// TIA Portal V21 export
FUNCTION_BLOCK "FB307"   // FB307, LAD
TITLE = FB307
{ S7_Optimized_Access := 'FALSE' }
AUTHOR : PRECISE
FAMILY : PRECISE
// RAW MATERIAL ADDITION MANUAL
// stored: AutoNumber false, SetENOAutomatically false
   VAR_INPUT
      Enable : Bool;
      Disable : Bool;
      Fault : Bool;
      SecPulse : Bool;
      AlwaysTrue : Bool;
      StartConfirmationPopupSel : Bool;   // StartConfirmationPopupSel: 0-NO/1-YES
      EndConfirmationPopupSel : Bool;   // EndConfirmationPopupSel: 0-NO/1-YES
      MixingTimerDone : Bool;
      SetRMNo : Int := 1;   // Max-10
      VesselSafetyPressure : Real;
      VesselActPressure : Real;
   END_VAR
   VAR_OUTPUT
      StartConfirmationPopup : Bool;   // For Start Confirmation Popup Selection: Yes
      EndConfirmationPopup : Bool;   // For End Confirmation Popup Selection: Yes
      RMAddPopup : Bool;
      VisibleRM1 : Bool;
      VisibleRM2 : Bool;
      VisibleRM3 : Bool;
      VisibleRM4 : Bool;
      VisibleRM5 : Bool;
      VisibleRM6 : Bool;
      VisibleRM7 : Bool;
      VisibleRM8 : Bool;
      VisibleRM9 : Bool;
      VisibleRM10 : Bool;
      PrintTrigger : Bool;
      MixerCmd : Bool;
      PrintWord : Int;
      PrintStatus : String[50];
      VesselUnderPressure : Bool;
   END_VAR
   VAR_IN_OUT
      Start : Bool;
      Stop : Bool;
      Reset : Bool;
      StartConfirmationAck : Bool;   // For Start Confirmation Popup Selection: Yes
      EndConfirmationAck : Bool;   // For End Confirmation Popup Selection: Yes
      AckRM1 : Bool;
      AckRM2 : Bool;
      AckRM3 : Bool;
      AckRM4 : Bool;
      AckRM5 : Bool;
      AckRM6 : Bool;
      AckRM7 : Bool;
      AckRM8 : Bool;
      AckRM9 : Bool;
      AckRM10 : Bool;
      Running : Bool;
      Selected : Bool;
      Paused : Bool;
      StartConfirmationPopupTemp : Bool;   // For Start Confirmation Popup Selection: Yes
      EndConfirmationPopupTemp : Bool;   // For End Confirmation Popup Selection: Yes
      RMAddStarted : Bool;
      RMAddOver : Bool;
      AddDoneRM1 : Bool;
      AddDoneRM2 : Bool;
      AddDoneRM3 : Bool;
      AddDoneRM4 : Bool;
      AddDoneRM5 : Bool;
      AddDoneRM6 : Bool;
      AddDoneRM7 : Bool;
      AddDoneRM8 : Bool;
      AddDoneRM9 : Bool;
      AddDoneRM10 : Bool;
   END_VAR
   VAR
      PrintTriggerTemp : Bool;
      RE1 : Bool;
      RE2 : Bool;
      RE3 : Bool;
      RE4 : Bool;
      RE5 : Bool;
      RE6 : Bool;
      RE7 : Bool;
      RE8 : Bool;
      RE9 : Bool;
      RE10 : Bool;
      RE11 : Bool;
      RE12 : Bool;
      RE13 : Bool;
      RE14 : Bool;
      RE15 : Bool;
      RE16 : Bool;
      RE17 : Bool;
      PrintTriggerResetTimer { S7_SetPoint := 'True'} : TON_TIME;
      BtnResetTimer { S7_SetPoint := 'True'} : TON_TIME;
      RMAddOverDelay { S7_SetPoint := 'True'} : TON_TIME;
      NameRM1 : String[100];
      NameRM2 : String[100];
      NameRM3 : String[100];
      NameRM4 : String[100];
      NameRM5 : String[100];
      NameRM6 : String[100];
      NameRM7 : String[100];
      NameRM8 : String[100];
      NameRM9 : String[100];
      NameRM10 : String[100];
   END_VAR
   VAR_TEMP
      STATUS1 : String[40];
      STATUS2 : String[40];
      STATUS3 : String[40];
      STATUS4 : String[40];
      STATUS5 : String[40];
      STATUS6 : String[40];
      STATUS7 : String[40];
      STATUS8 : String[40];
      STATUS9 : String[40];
      STATUS10 : String[40];
      Blank : String[40];
   END_VAR
   VAR_TEMP   // added for the SCL form of the ladder/FBD networks
      _w1 : Bool;
      _w2 : Bool;
      _w3 : Bool;
      _w4 : Bool;
      _w5 : Bool;
      _w6 : Bool;
      _w7 : Bool;
      _w8 : Bool;
      _w9 : Bool;
      _w10 : Bool;
      _w11 : Bool;
      _w12 : Bool;
      _w13 : Bool;
      _w14 : Bool;
      _w15 : Bool;
      _w16 : Bool;
      _w17 : Bool;
      _w18 : Bool;
      _w19 : Bool;
      _w20 : Bool;
      _w21 : Bool;
      _w22 : Bool;
      _w23 : Bool;
      _w24 : Bool;
      _w25 : Bool;
   END_VAR
BEGIN

REGION Network 1: Running
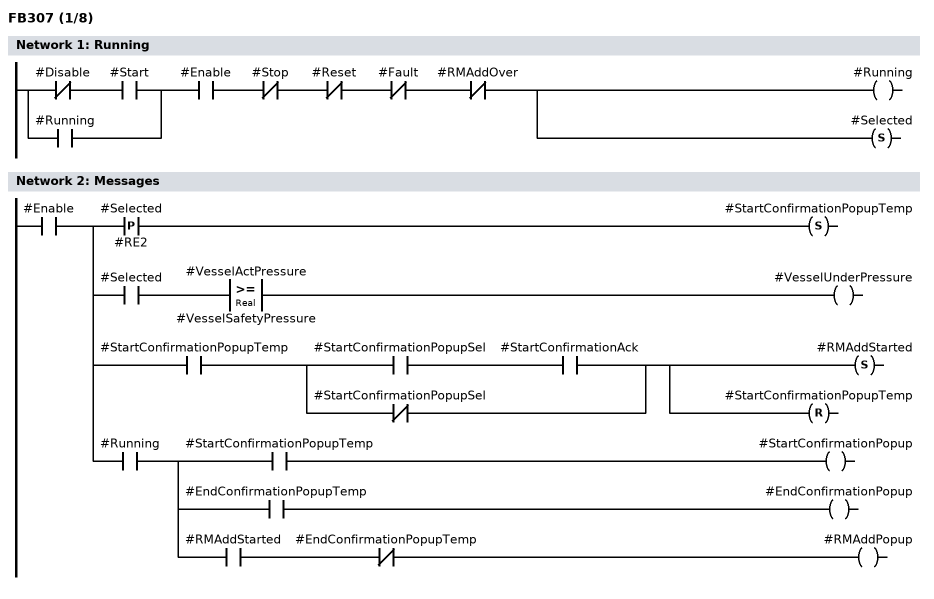
   RUNG wire#powerrail
      I_Contact( #Disable )
      Contact( #Start )
      wire#w1
      Contact( #Enable )
      I_Contact( #Stop )
      I_Contact( #Reset )
      I_Contact( #Fault )
      I_Contact( #RMAddOver )
      wire#w2
      Coil( #Running )
   END_RUNG
   RUNG wire#powerrail
      Contact( #Running )
   END_RUNG wire#w1
   RUNG wire#w2
      S_Coil( #Selected )
   END_RUNG
   // the same network as SCL:
   #Running := ((NOT #Disable AND #Start) OR #Running) AND #Enable AND NOT #Stop AND NOT #Reset AND NOT #Fault AND NOT #RMAddOver;
   IF #Running THEN #Selected := TRUE; END_IF;
END_REGION

REGION Network 2: Messages
   RUNG wire#powerrail
      Contact( #Enable )
      wire#w1
      P_Contact(operand := #Selected, bit := #RE2)
      S_Coil( #StartConfirmationPopupTemp )
   END_RUNG
   RUNG wire#w1
      Contact( #Selected )
      { S7_Templates := "SrcType := Real" } GE_Contact(in1 := #VesselActPressure, in2 := #VesselSafetyPressure)
      Coil( #VesselUnderPressure )
   END_RUNG
   RUNG wire#w1
      Contact( #StartConfirmationPopupTemp )
      wire#w2
      Contact( #StartConfirmationPopupSel )
      Contact( #StartConfirmationAck )
      wire#w3
      S_Coil( #RMAddStarted )
   END_RUNG
   RUNG wire#w2
      I_Contact( #StartConfirmationPopupSel )
   END_RUNG wire#w3
   RUNG wire#w3
      R_Coil( #StartConfirmationPopupTemp )
   END_RUNG
   RUNG wire#w1
      Contact( #Running )
      wire#w4
      Contact( #StartConfirmationPopupTemp )
      Coil( #StartConfirmationPopup )
   END_RUNG
   RUNG wire#w4
      Contact( #EndConfirmationPopupTemp )
      Coil( #EndConfirmationPopup )
   END_RUNG
   RUNG wire#w4
      Contact( #RMAddStarted )
      I_Contact( #EndConfirmationPopupTemp )
      Coil( #RMAddPopup )
   END_RUNG
   // the same network as SCL:
   #_w1 := #Enable AND #Selected AND NOT #RE2;   // rising edge of #Selected
   #RE2 := #Selected;
   IF #_w1 THEN #StartConfirmationPopupTemp := TRUE; END_IF;
   #VesselUnderPressure := #Enable AND #Selected AND (#VesselActPressure >= #VesselSafetyPressure);
   IF #Enable AND #StartConfirmationPopupTemp AND ((#StartConfirmationPopupSel AND #StartConfirmationAck) OR NOT #StartConfirmationPopupSel) THEN
       #RMAddStarted := TRUE;
       #StartConfirmationPopupTemp := FALSE;
   END_IF;
   #_w2 := #Enable AND #Running;
   #StartConfirmationPopup := #_w2 AND #StartConfirmationPopupTemp;
   #EndConfirmationPopup := #_w2 AND #EndConfirmationPopupTemp;
   #RMAddPopup := #_w2 AND #RMAddStarted AND NOT #EndConfirmationPopupTemp;
END_REGION

REGION Network 3: Visibility for RM
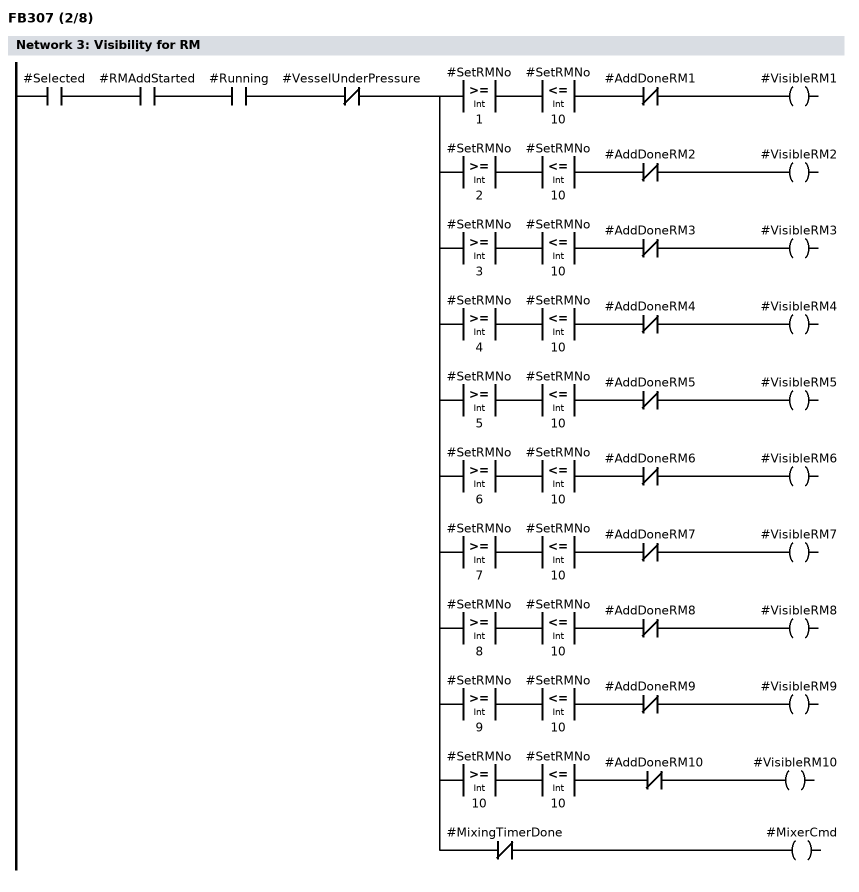
   RUNG wire#powerrail
      Contact( #Selected )
      Contact( #RMAddStarted )
      Contact( #Running )
      I_Contact( #VesselUnderPressure )
      wire#w1
      { S7_Templates := "SrcType := Int" } GE_Contact(in1 := #SetRMNo, in2 := 1)
      { S7_Templates := "SrcType := Int" } LE_Contact(in1 := #SetRMNo, in2 := 10)
      I_Contact( #AddDoneRM1 )
      Coil( #VisibleRM1 )
   END_RUNG
   RUNG wire#w1
      { S7_Templates := "SrcType := Int" } GE_Contact(in1 := #SetRMNo, in2 := 2)
      { S7_Templates := "SrcType := Int" } LE_Contact(in1 := #SetRMNo, in2 := 10)
      I_Contact( #AddDoneRM2 )
      Coil( #VisibleRM2 )
   END_RUNG
   RUNG wire#w1
      { S7_Templates := "SrcType := Int" } GE_Contact(in1 := #SetRMNo, in2 := 3)
      { S7_Templates := "SrcType := Int" } LE_Contact(in1 := #SetRMNo, in2 := 10)
      I_Contact( #AddDoneRM3 )
      Coil( #VisibleRM3 )
   END_RUNG
   RUNG wire#w1
      { S7_Templates := "SrcType := Int" } GE_Contact(in1 := #SetRMNo, in2 := 4)
      { S7_Templates := "SrcType := Int" } LE_Contact(in1 := #SetRMNo, in2 := 10)
      I_Contact( #AddDoneRM4 )
      Coil( #VisibleRM4 )
   END_RUNG
   RUNG wire#w1
      { S7_Templates := "SrcType := Int" } GE_Contact(in1 := #SetRMNo, in2 := 5)
      { S7_Templates := "SrcType := Int" } LE_Contact(in1 := #SetRMNo, in2 := 10)
      I_Contact( #AddDoneRM5 )
      Coil( #VisibleRM5 )
   END_RUNG
   RUNG wire#w1
      { S7_Templates := "SrcType := Int" } GE_Contact(in1 := #SetRMNo, in2 := 6)
      { S7_Templates := "SrcType := Int" } LE_Contact(in1 := #SetRMNo, in2 := 10)
      I_Contact( #AddDoneRM6 )
      Coil( #VisibleRM6 )
   END_RUNG
   RUNG wire#w1
      { S7_Templates := "SrcType := Int" } GE_Contact(in1 := #SetRMNo, in2 := 7)
      { S7_Templates := "SrcType := Int" } LE_Contact(in1 := #SetRMNo, in2 := 10)
      I_Contact( #AddDoneRM7 )
      Coil( #VisibleRM7 )
   END_RUNG
   RUNG wire#w1
      { S7_Templates := "SrcType := Int" } GE_Contact(in1 := #SetRMNo, in2 := 8)
      { S7_Templates := "SrcType := Int" } LE_Contact(in1 := #SetRMNo, in2 := 10)
      I_Contact( #AddDoneRM8 )
      Coil( #VisibleRM8 )
   END_RUNG
   RUNG wire#w1
      { S7_Templates := "SrcType := Int" } GE_Contact(in1 := #SetRMNo, in2 := 9)
      { S7_Templates := "SrcType := Int" } LE_Contact(in1 := #SetRMNo, in2 := 10)
      I_Contact( #AddDoneRM9 )
      Coil( #VisibleRM9 )
   END_RUNG
   RUNG wire#w1
      { S7_Templates := "SrcType := Int" } GE_Contact(in1 := #SetRMNo, in2 := 10)
      { S7_Templates := "SrcType := Int" } LE_Contact(in1 := #SetRMNo, in2 := 10)
      I_Contact( #AddDoneRM10 )
      Coil( #VisibleRM10 )
   END_RUNG
   RUNG wire#w1
      I_Contact( #MixingTimerDone )
      Coil( #MixerCmd )
   END_RUNG
   // the same network as SCL:
   #_w1 := #Selected AND #RMAddStarted AND #Running AND NOT #VesselUnderPressure;
   #VisibleRM1 := #_w1 AND (#SetRMNo >= 1) AND (#SetRMNo <= 10) AND NOT #AddDoneRM1;
   #VisibleRM2 := #_w1 AND (#SetRMNo >= 2) AND (#SetRMNo <= 10) AND NOT #AddDoneRM2;
   #VisibleRM3 := #_w1 AND (#SetRMNo >= 3) AND (#SetRMNo <= 10) AND NOT #AddDoneRM3;
   #VisibleRM4 := #_w1 AND (#SetRMNo >= 4) AND (#SetRMNo <= 10) AND NOT #AddDoneRM4;
   #VisibleRM5 := #_w1 AND (#SetRMNo >= 5) AND (#SetRMNo <= 10) AND NOT #AddDoneRM5;
   #VisibleRM6 := #_w1 AND (#SetRMNo >= 6) AND (#SetRMNo <= 10) AND NOT #AddDoneRM6;
   #VisibleRM7 := #_w1 AND (#SetRMNo >= 7) AND (#SetRMNo <= 10) AND NOT #AddDoneRM7;
   #VisibleRM8 := #_w1 AND (#SetRMNo >= 8) AND (#SetRMNo <= 10) AND NOT #AddDoneRM8;
   #VisibleRM9 := #_w1 AND (#SetRMNo >= 9) AND (#SetRMNo <= 10) AND NOT #AddDoneRM9;
   #VisibleRM10 := #_w1 AND (#SetRMNo >= 10) AND (#SetRMNo <= 10) AND NOT #AddDoneRM10;
   #MixerCmd := #_w1 AND NOT #MixingTimerDone;
END_REGION

REGION Network 4: Add Done
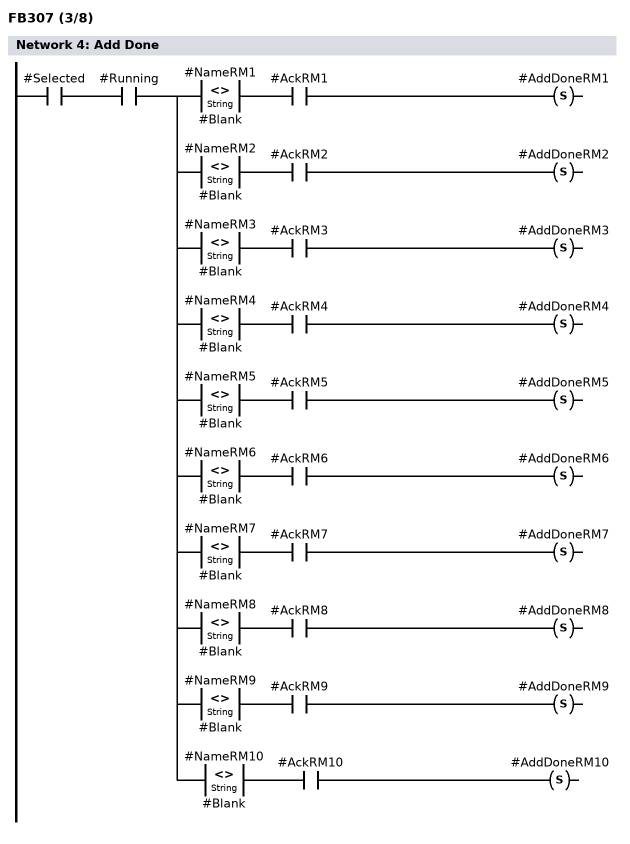
   RUNG wire#powerrail
      Contact( #Selected )
      Contact( #Running )
      wire#w1
      { S7_Templates := "SrcType := String" } NE_Contact(in1 := #NameRM1, in2 := #Blank)
      Contact( #AckRM1 )
      S_Coil( #AddDoneRM1 )
   END_RUNG
   RUNG wire#w1
      { S7_Templates := "SrcType := String" } NE_Contact(in1 := #NameRM2, in2 := #Blank)
      Contact( #AckRM2 )
      S_Coil( #AddDoneRM2 )
   END_RUNG
   RUNG wire#w1
      { S7_Templates := "SrcType := String" } NE_Contact(in1 := #NameRM3, in2 := #Blank)
      Contact( #AckRM3 )
      S_Coil( #AddDoneRM3 )
   END_RUNG
   RUNG wire#w1
      { S7_Templates := "SrcType := String" } NE_Contact(in1 := #NameRM4, in2 := #Blank)
      Contact( #AckRM4 )
      S_Coil( #AddDoneRM4 )
   END_RUNG
   RUNG wire#w1
      { S7_Templates := "SrcType := String" } NE_Contact(in1 := #NameRM5, in2 := #Blank)
      Contact( #AckRM5 )
      S_Coil( #AddDoneRM5 )
   END_RUNG
   RUNG wire#w1
      { S7_Templates := "SrcType := String" } NE_Contact(in1 := #NameRM6, in2 := #Blank)
      Contact( #AckRM6 )
      S_Coil( #AddDoneRM6 )
   END_RUNG
   RUNG wire#w1
      { S7_Templates := "SrcType := String" } NE_Contact(in1 := #NameRM7, in2 := #Blank)
      Contact( #AckRM7 )
      S_Coil( #AddDoneRM7 )
   END_RUNG
   RUNG wire#w1
      { S7_Templates := "SrcType := String" } NE_Contact(in1 := #NameRM8, in2 := #Blank)
      Contact( #AckRM8 )
      S_Coil( #AddDoneRM8 )
   END_RUNG
   RUNG wire#w1
      { S7_Templates := "SrcType := String" } NE_Contact(in1 := #NameRM9, in2 := #Blank)
      Contact( #AckRM9 )
      S_Coil( #AddDoneRM9 )
   END_RUNG
   RUNG wire#w1
      { S7_Templates := "SrcType := String" } NE_Contact(in1 := #NameRM10, in2 := #Blank)
      Contact( #AckRM10 )
      S_Coil( #AddDoneRM10 )
   END_RUNG
   // the same network as SCL:
   #_w1 := #Selected AND #Running;
   IF #_w1 AND (#NameRM1 <> #Blank) AND #AckRM1 THEN #AddDoneRM1 := TRUE; END_IF;
   IF #_w1 AND (#NameRM2 <> #Blank) AND #AckRM2 THEN #AddDoneRM2 := TRUE; END_IF;
   IF #_w1 AND (#NameRM3 <> #Blank) AND #AckRM3 THEN #AddDoneRM3 := TRUE; END_IF;
   IF #_w1 AND (#NameRM4 <> #Blank) AND #AckRM4 THEN #AddDoneRM4 := TRUE; END_IF;
   IF #_w1 AND (#NameRM5 <> #Blank) AND #AckRM5 THEN #AddDoneRM5 := TRUE; END_IF;
   IF #_w1 AND (#NameRM6 <> #Blank) AND #AckRM6 THEN #AddDoneRM6 := TRUE; END_IF;
   IF #_w1 AND (#NameRM7 <> #Blank) AND #AckRM7 THEN #AddDoneRM7 := TRUE; END_IF;
   IF #_w1 AND (#NameRM8 <> #Blank) AND #AckRM8 THEN #AddDoneRM8 := TRUE; END_IF;
   IF #_w1 AND (#NameRM9 <> #Blank) AND #AckRM9 THEN #AddDoneRM9 := TRUE; END_IF;
   IF #_w1 AND (#NameRM10 <> #Blank) AND #AckRM10 THEN #AddDoneRM10 := TRUE; END_IF;
END_REGION

REGION Network 5: All Addition Done
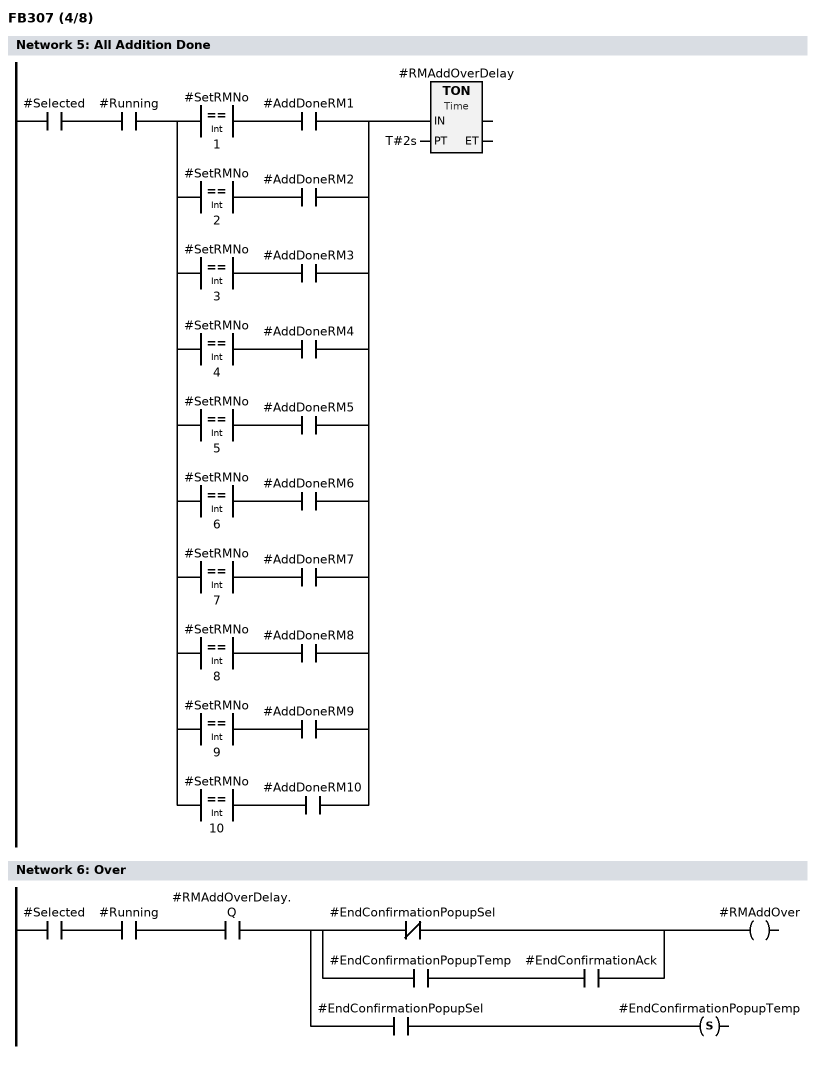
   RUNG wire#powerrail
      Contact( #Selected )
      Contact( #Running )
      wire#w1
      { S7_Templates := "SrcType := Int" } EQ_Contact(in1 := #SetRMNo, in2 := 1)
      Contact( #AddDoneRM1 )
      wire#w2
      { S7_Templates := "time_type := Time" } #RMAddOverDelay.TON(pt := T#2s, et =>)
   END_RUNG
   RUNG wire#w1
      { S7_Templates := "SrcType := Int" } EQ_Contact(in1 := #SetRMNo, in2 := 2)
      Contact( #AddDoneRM2 )
   END_RUNG wire#w2
   RUNG wire#w1
      { S7_Templates := "SrcType := Int" } EQ_Contact(in1 := #SetRMNo, in2 := 3)
      Contact( #AddDoneRM3 )
   END_RUNG wire#w2
   RUNG wire#w1
      { S7_Templates := "SrcType := Int" } EQ_Contact(in1 := #SetRMNo, in2 := 4)
      Contact( #AddDoneRM4 )
   END_RUNG wire#w2
   RUNG wire#w1
      { S7_Templates := "SrcType := Int" } EQ_Contact(in1 := #SetRMNo, in2 := 5)
      Contact( #AddDoneRM5 )
   END_RUNG wire#w2
   RUNG wire#w1
      { S7_Templates := "SrcType := Int" } EQ_Contact(in1 := #SetRMNo, in2 := 6)
      Contact( #AddDoneRM6 )
   END_RUNG wire#w2
   RUNG wire#w1
      { S7_Templates := "SrcType := Int" } EQ_Contact(in1 := #SetRMNo, in2 := 7)
      Contact( #AddDoneRM7 )
   END_RUNG wire#w2
   RUNG wire#w1
      { S7_Templates := "SrcType := Int" } EQ_Contact(in1 := #SetRMNo, in2 := 8)
      Contact( #AddDoneRM8 )
   END_RUNG wire#w2
   RUNG wire#w1
      { S7_Templates := "SrcType := Int" } EQ_Contact(in1 := #SetRMNo, in2 := 9)
      Contact( #AddDoneRM9 )
   END_RUNG wire#w2
   RUNG wire#w1
      { S7_Templates := "SrcType := Int" } EQ_Contact(in1 := #SetRMNo, in2 := 10)
      Contact( #AddDoneRM10 )
   END_RUNG wire#w2
   // the same network as SCL:
   #RMAddOverDelay(IN := #Selected AND #Running AND (((#SetRMNo = 1) AND #AddDoneRM1) OR ((#SetRMNo = 2) AND #AddDoneRM2) OR ((#SetRMNo = 3) AND #AddDoneRM3) OR ((#SetRMNo = 4) AND #AddDoneRM4) OR ((#SetRMNo = 5) AND #AddDoneRM5) OR ((#SetRMNo = 6) AND #AddDoneRM6) OR ((#SetRMNo = 7) AND #AddDoneRM7) OR ((#SetRMNo = 8) AND #AddDoneRM8) OR ((#SetRMNo = 9) AND #AddDoneRM9) OR ((#SetRMNo = 10) AND #AddDoneRM10)),   // TON
                   PT := T#2s);
END_REGION

REGION Network 6: Over
   RUNG wire#powerrail
      Contact( #Selected )
      Contact( #Running )
      Contact( #RMAddOverDelay.Q )
      wire#w1
      I_Contact( #EndConfirmationPopupSel )
      wire#w2
      Coil( #RMAddOver )
   END_RUNG
   RUNG wire#w1
      Contact( #EndConfirmationPopupTemp )
      Contact( #EndConfirmationAck )
   END_RUNG wire#w2
   RUNG wire#w1
      Contact( #EndConfirmationPopupSel )
      S_Coil( #EndConfirmationPopupTemp )
   END_RUNG
   // the same network as SCL:
   #_w1 := #Selected AND #Running AND #RMAddOverDelay.Q;
   #RMAddOver := #_w1 AND (NOT #EndConfirmationPopupSel OR (#EndConfirmationPopupTemp AND #EndConfirmationAck));
   IF #_w1 AND #EndConfirmationPopupSel THEN #EndConfirmationPopupTemp := TRUE; END_IF;
END_REGION

REGION Network 7: Event Status
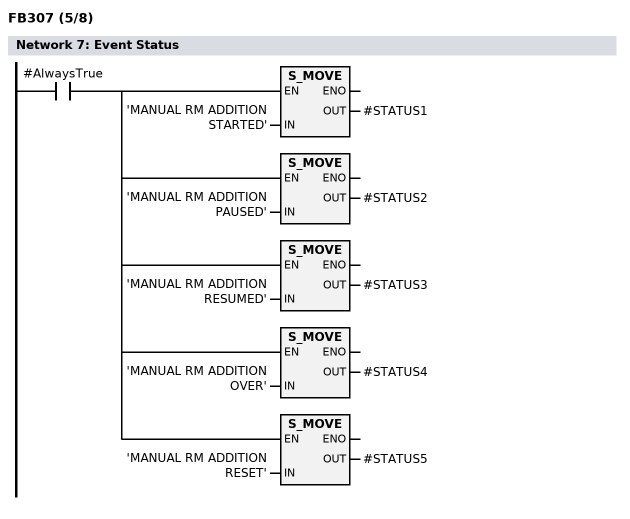
   RUNG wire#powerrail
      Contact( #AlwaysTrue )
      wire#w1
      S_Move(in := 'MANUAL RM ADDITION STARTED', out => #STATUS1)
   END_RUNG
   RUNG wire#w1
      S_Move(in := 'MANUAL RM ADDITION PAUSED', out => #STATUS2)
   END_RUNG
   RUNG wire#w1
      S_Move(in := 'MANUAL RM ADDITION RESUMED', out => #STATUS3)
   END_RUNG
   RUNG wire#w1
      S_Move(in := 'MANUAL RM ADDITION OVER', out => #STATUS4)
   END_RUNG
   RUNG wire#w1
      S_Move(in := 'MANUAL RM ADDITION RESET', out => #STATUS5)
   END_RUNG
   // the same network as SCL:
   IF #AlwaysTrue THEN
       #STATUS1 := 'MANUAL RM ADDITION STARTED';
       #STATUS2 := 'MANUAL RM ADDITION PAUSED';
       #STATUS3 := 'MANUAL RM ADDITION RESUMED';
       #STATUS4 := 'MANUAL RM ADDITION OVER';
       #STATUS5 := 'MANUAL RM ADDITION RESET';
   END_IF;
END_REGION

REGION Network 8: Print Logic
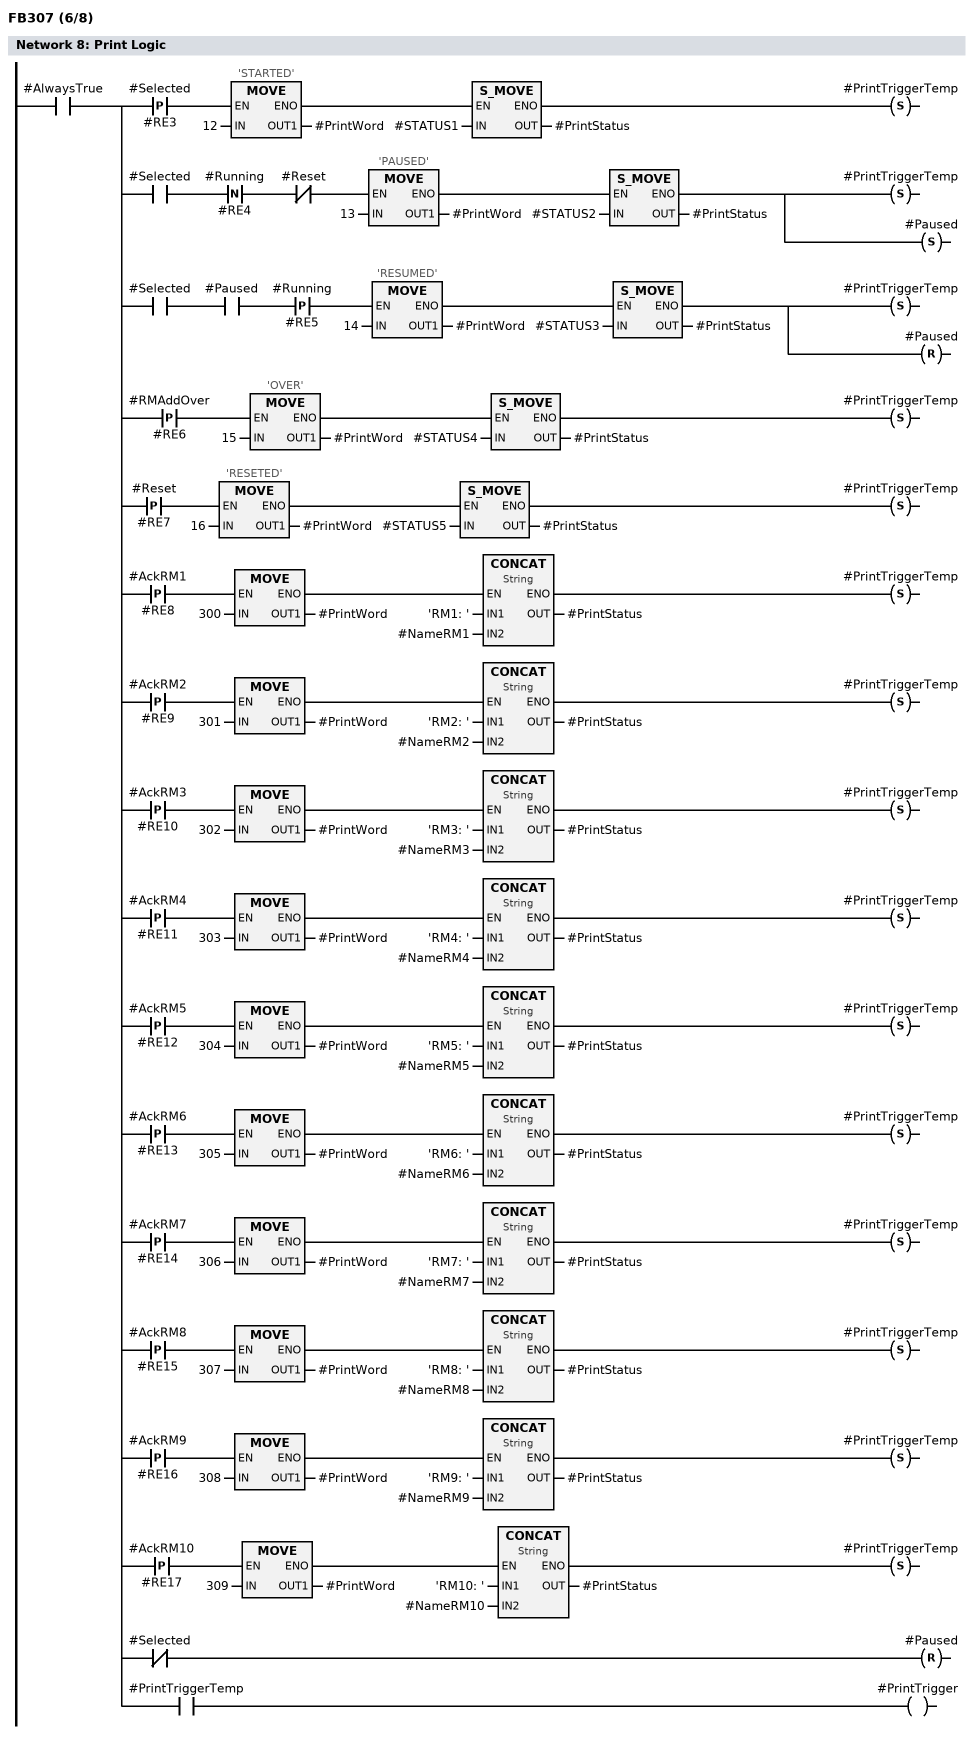
   RUNG wire#powerrail
      Contact( #AlwaysTrue )
      wire#w1
      P_Contact(operand := #Selected, bit := #RE3)
      { S7_GenerateENO := "TRUE" } Move(in := 12, out1 => #PrintWord)   // 'STARTED'
      S_Move(in := #STATUS1, out => #PrintStatus)
      S_Coil( #PrintTriggerTemp )
   END_RUNG
   RUNG wire#w1
      Contact( #Selected )
      N_Contact(operand := #Running, bit := #RE4)
      I_Contact( #Reset )
      { S7_GenerateENO := "TRUE" } Move(in := 13, out1 => #PrintWord)   // 'PAUSED'
      S_Move(in := #STATUS2, out => #PrintStatus)
      wire#w2
      S_Coil( #PrintTriggerTemp )
   END_RUNG
   RUNG wire#w2
      S_Coil( #Paused )
   END_RUNG
   RUNG wire#w1
      Contact( #Selected )
      Contact( #Paused )
      P_Contact(operand := #Running, bit := #RE5)
      { S7_GenerateENO := "TRUE" } Move(in := 14, out1 => #PrintWord)   // 'RESUMED'
      S_Move(in := #STATUS3, out => #PrintStatus)
      wire#w3
      S_Coil( #PrintTriggerTemp )
   END_RUNG
   RUNG wire#w3
      R_Coil( #Paused )
   END_RUNG
   RUNG wire#w1
      P_Contact(operand := #RMAddOver, bit := #RE6)
      { S7_GenerateENO := "TRUE" } Move(in := 15, out1 => #PrintWord)   // 'OVER'
      S_Move(in := #STATUS4, out => #PrintStatus)
      S_Coil( #PrintTriggerTemp )
   END_RUNG
   RUNG wire#w1
      P_Contact(operand := #Reset, bit := #RE7)
      { S7_GenerateENO := "TRUE" } Move(in := 16, out1 => #PrintWord)   // 'RESETED'
      S_Move(in := #STATUS5, out => #PrintStatus)
      S_Coil( #PrintTriggerTemp )
   END_RUNG
   RUNG wire#w1
      P_Contact(operand := #AckRM1, bit := #RE8)
      { S7_GenerateENO := "TRUE" } Move(in := 300, out1 => #PrintWord)
      { S7_Templates := "[card := 2, str_type := String]" } CONCAT(IN1 := 'RM1: ', IN2 := #NameRM1, OUT => #PrintStatus)
      S_Coil( #PrintTriggerTemp )
   END_RUNG
   RUNG wire#w1
      P_Contact(operand := #AckRM2, bit := #RE9)
      { S7_GenerateENO := "TRUE" } Move(in := 301, out1 => #PrintWord)
      { S7_Templates := "[card := 2, str_type := String]" } CONCAT(IN1 := 'RM2: ', IN2 := #NameRM2, OUT => #PrintStatus)
      S_Coil( #PrintTriggerTemp )
   END_RUNG
   RUNG wire#w1
      P_Contact(operand := #AckRM3, bit := #RE10)
      { S7_GenerateENO := "TRUE" } Move(in := 302, out1 => #PrintWord)
      { S7_Templates := "[card := 2, str_type := String]" } CONCAT(IN1 := 'RM3: ', IN2 := #NameRM3, OUT => #PrintStatus)
      S_Coil( #PrintTriggerTemp )
   END_RUNG
   RUNG wire#w1
      P_Contact(operand := #AckRM4, bit := #RE11)
      { S7_GenerateENO := "TRUE" } Move(in := 303, out1 => #PrintWord)
      { S7_Templates := "[card := 2, str_type := String]" } CONCAT(IN1 := 'RM4: ', IN2 := #NameRM4, OUT => #PrintStatus)
      S_Coil( #PrintTriggerTemp )
   END_RUNG
   RUNG wire#w1
      P_Contact(operand := #AckRM5, bit := #RE12)
      { S7_GenerateENO := "TRUE" } Move(in := 304, out1 => #PrintWord)
      { S7_Templates := "[card := 2, str_type := String]" } CONCAT(IN1 := 'RM5: ', IN2 := #NameRM5, OUT => #PrintStatus)
      S_Coil( #PrintTriggerTemp )
   END_RUNG
   RUNG wire#w1
      P_Contact(operand := #AckRM6, bit := #RE13)
      { S7_GenerateENO := "TRUE" } Move(in := 305, out1 => #PrintWord)
      { S7_Templates := "[card := 2, str_type := String]" } CONCAT(IN1 := 'RM6: ', IN2 := #NameRM6, OUT => #PrintStatus)
      S_Coil( #PrintTriggerTemp )
   END_RUNG
   RUNG wire#w1
      P_Contact(operand := #AckRM7, bit := #RE14)
      { S7_GenerateENO := "TRUE" } Move(in := 306, out1 => #PrintWord)
      { S7_Templates := "[card := 2, str_type := String]" } CONCAT(IN1 := 'RM7: ', IN2 := #NameRM7, OUT => #PrintStatus)
      S_Coil( #PrintTriggerTemp )
   END_RUNG
   RUNG wire#w1
      P_Contact(operand := #AckRM8, bit := #RE15)
      { S7_GenerateENO := "TRUE" } Move(in := 307, out1 => #PrintWord)
      { S7_Templates := "[card := 2, str_type := String]" } CONCAT(IN1 := 'RM8: ', IN2 := #NameRM8, OUT => #PrintStatus)
      S_Coil( #PrintTriggerTemp )
   END_RUNG
   RUNG wire#w1
      P_Contact(operand := #AckRM9, bit := #RE16)
      { S7_GenerateENO := "TRUE" } Move(in := 308, out1 => #PrintWord)
      { S7_Templates := "[card := 2, str_type := String]" } CONCAT(IN1 := 'RM9: ', IN2 := #NameRM9, OUT => #PrintStatus)
      S_Coil( #PrintTriggerTemp )
   END_RUNG
   RUNG wire#w1
      P_Contact(operand := #AckRM10, bit := #RE17)
      { S7_GenerateENO := "TRUE" } Move(in := 309, out1 => #PrintWord)
      { S7_Templates := "[card := 2, str_type := String]" } CONCAT(IN1 := 'RM10: ', IN2 := #NameRM10, OUT => #PrintStatus)
      S_Coil( #PrintTriggerTemp )
   END_RUNG
   RUNG wire#w1
      I_Contact( #Selected )
      R_Coil( #Paused )
   END_RUNG
   RUNG wire#w1
      Contact( #PrintTriggerTemp )
      Coil( #PrintTrigger )
   END_RUNG
   // the same network as SCL:
   // ENO of a box is taken as its EN; it also drops when the box reports an error
   #_w1 := #AlwaysTrue AND #Selected AND NOT #RE3;   // rising edge of #Selected
   #RE3 := #Selected;
   IF #_w1 THEN
       #PrintWord := 12;   // 'STARTED'
       #PrintStatus := #STATUS1;
       #PrintTriggerTemp := TRUE;
   END_IF;
   #_w2 := #AlwaysTrue AND #Selected AND NOT #Running AND #RE4;   // falling edge of #Running
   #RE4 := #Running;
   IF #_w2 AND NOT #Reset THEN
       #PrintWord := 13;   // 'PAUSED'
       #PrintStatus := #STATUS2;
       #PrintTriggerTemp := TRUE;
       #Paused := TRUE;
   END_IF;
   #_w3 := #AlwaysTrue AND #Selected AND #Paused AND #Running AND NOT #RE5;   // rising edge of #Running
   #RE5 := #Running;
   IF #_w3 THEN
       #PrintWord := 14;   // 'RESUMED'
       #PrintStatus := #STATUS3;
       #PrintTriggerTemp := TRUE;
       #Paused := FALSE;
   END_IF;
   #_w4 := #AlwaysTrue AND #RMAddOver AND NOT #RE6;   // rising edge of #RMAddOver
   #RE6 := #RMAddOver;
   IF #_w4 THEN
       #PrintWord := 15;   // 'OVER'
       #PrintStatus := #STATUS4;
       #PrintTriggerTemp := TRUE;
   END_IF;
   #_w5 := #AlwaysTrue AND #Reset AND NOT #RE7;   // rising edge of #Reset
   #RE7 := #Reset;
   IF #_w5 THEN
       #PrintWord := 16;   // 'RESETED'
       #PrintStatus := #STATUS5;
       #PrintTriggerTemp := TRUE;
   END_IF;
   #_w6 := #AlwaysTrue AND #AckRM1 AND NOT #RE8;   // rising edge of #AckRM1
   #RE8 := #AckRM1;
   IF #_w6 THEN #PrintWord := 300; END_IF;
   CONCAT(EN := #_w6, IN1 := 'RM1: ', IN2 := #NameRM1, OUT => #PrintStatus, ENO => #_w7);
   IF #_w7 THEN #PrintTriggerTemp := TRUE; END_IF;
   #_w8 := #AlwaysTrue AND #AckRM2 AND NOT #RE9;   // rising edge of #AckRM2
   #RE9 := #AckRM2;
   IF #_w8 THEN #PrintWord := 301; END_IF;
   CONCAT(EN := #_w8, IN1 := 'RM2: ', IN2 := #NameRM2, OUT => #PrintStatus, ENO => #_w9);
   IF #_w9 THEN #PrintTriggerTemp := TRUE; END_IF;
   #_w10 := #AlwaysTrue AND #AckRM3 AND NOT #RE10;   // rising edge of #AckRM3
   #RE10 := #AckRM3;
   IF #_w10 THEN #PrintWord := 302; END_IF;
   CONCAT(EN := #_w10, IN1 := 'RM3: ', IN2 := #NameRM3, OUT => #PrintStatus, ENO => #_w11);
   IF #_w11 THEN #PrintTriggerTemp := TRUE; END_IF;
   #_w12 := #AlwaysTrue AND #AckRM4 AND NOT #RE11;   // rising edge of #AckRM4
   #RE11 := #AckRM4;
   IF #_w12 THEN #PrintWord := 303; END_IF;
   CONCAT(EN := #_w12, IN1 := 'RM4: ', IN2 := #NameRM4, OUT => #PrintStatus, ENO => #_w13);
   IF #_w13 THEN #PrintTriggerTemp := TRUE; END_IF;
   #_w14 := #AlwaysTrue AND #AckRM5 AND NOT #RE12;   // rising edge of #AckRM5
   #RE12 := #AckRM5;
   IF #_w14 THEN #PrintWord := 304; END_IF;
   CONCAT(EN := #_w14, IN1 := 'RM5: ', IN2 := #NameRM5, OUT => #PrintStatus, ENO => #_w15);
   IF #_w15 THEN #PrintTriggerTemp := TRUE; END_IF;
   #_w16 := #AlwaysTrue AND #AckRM6 AND NOT #RE13;   // rising edge of #AckRM6
   #RE13 := #AckRM6;
   IF #_w16 THEN #PrintWord := 305; END_IF;
   CONCAT(EN := #_w16, IN1 := 'RM6: ', IN2 := #NameRM6, OUT => #PrintStatus, ENO => #_w17);
   IF #_w17 THEN #PrintTriggerTemp := TRUE; END_IF;
   #_w18 := #AlwaysTrue AND #AckRM7 AND NOT #RE14;   // rising edge of #AckRM7
   #RE14 := #AckRM7;
   IF #_w18 THEN #PrintWord := 306; END_IF;
   CONCAT(EN := #_w18, IN1 := 'RM7: ', IN2 := #NameRM7, OUT => #PrintStatus, ENO => #_w19);
   IF #_w19 THEN #PrintTriggerTemp := TRUE; END_IF;
   #_w20 := #AlwaysTrue AND #AckRM8 AND NOT #RE15;   // rising edge of #AckRM8
   #RE15 := #AckRM8;
   IF #_w20 THEN #PrintWord := 307; END_IF;
   CONCAT(EN := #_w20, IN1 := 'RM8: ', IN2 := #NameRM8, OUT => #PrintStatus, ENO => #_w21);
   IF #_w21 THEN #PrintTriggerTemp := TRUE; END_IF;
   #_w22 := #AlwaysTrue AND #AckRM9 AND NOT #RE16;   // rising edge of #AckRM9
   #RE16 := #AckRM9;
   IF #_w22 THEN #PrintWord := 308; END_IF;
   CONCAT(EN := #_w22, IN1 := 'RM9: ', IN2 := #NameRM9, OUT => #PrintStatus, ENO => #_w23);
   IF #_w23 THEN #PrintTriggerTemp := TRUE; END_IF;
   #_w24 := #AlwaysTrue AND #AckRM10 AND NOT #RE17;   // rising edge of #AckRM10
   #RE17 := #AckRM10;
   IF #_w24 THEN #PrintWord := 309; END_IF;
   CONCAT(EN := #_w24, IN1 := 'RM10: ', IN2 := #NameRM10, OUT => #PrintStatus, ENO => #_w25);
   IF #_w25 THEN #PrintTriggerTemp := TRUE; END_IF;
   IF #AlwaysTrue AND NOT #Selected THEN #Paused := FALSE; END_IF;
   #PrintTrigger := #AlwaysTrue AND #PrintTriggerTemp;
END_REGION

REGION Network 9: Print Trigger Reset
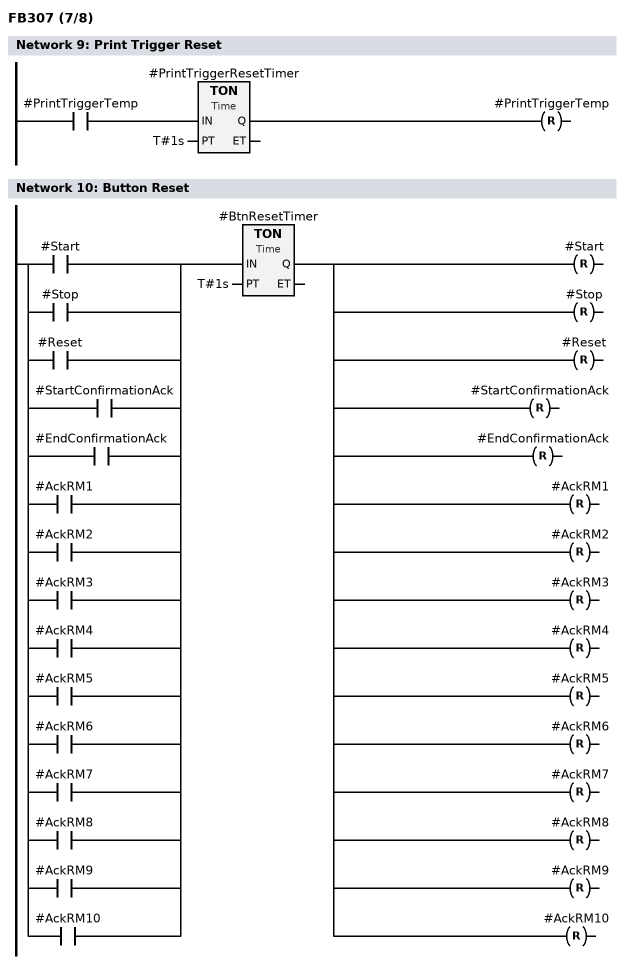
   RUNG wire#powerrail
      Contact( #PrintTriggerTemp )
      { S7_Templates := "time_type := Time" } #PrintTriggerResetTimer.TON(pt := T#1s, et =>)
      R_Coil( #PrintTriggerTemp )
   END_RUNG
   // the same network as SCL:
   #PrintTriggerResetTimer(IN := #PrintTriggerTemp, PT := T#1s);   // TON
   IF #PrintTriggerResetTimer.Q THEN #PrintTriggerTemp := FALSE; END_IF;
END_REGION

REGION Network 10: Button Reset
   RUNG wire#powerrail
      Contact( #Start )
      wire#w1
      { S7_Templates := "time_type := Time" } #BtnResetTimer.TON(pt := T#1s, et =>)
      wire#w2
      R_Coil( #Start )
   END_RUNG
   RUNG wire#powerrail
      Contact( #Stop )
   END_RUNG wire#w1
   RUNG wire#powerrail
      Contact( #Reset )
   END_RUNG wire#w1
   RUNG wire#powerrail
      Contact( #StartConfirmationAck )
   END_RUNG wire#w1
   RUNG wire#powerrail
      Contact( #EndConfirmationAck )
   END_RUNG wire#w1
   RUNG wire#powerrail
      Contact( #AckRM1 )
   END_RUNG wire#w1
   RUNG wire#powerrail
      Contact( #AckRM2 )
   END_RUNG wire#w1
   RUNG wire#powerrail
      Contact( #AckRM3 )
   END_RUNG wire#w1
   RUNG wire#powerrail
      Contact( #AckRM4 )
   END_RUNG wire#w1
   RUNG wire#powerrail
      Contact( #AckRM5 )
   END_RUNG wire#w1
   RUNG wire#powerrail
      Contact( #AckRM6 )
   END_RUNG wire#w1
   RUNG wire#powerrail
      Contact( #AckRM7 )
   END_RUNG wire#w1
   RUNG wire#powerrail
      Contact( #AckRM8 )
   END_RUNG wire#w1
   RUNG wire#powerrail
      Contact( #AckRM9 )
   END_RUNG wire#w1
   RUNG wire#powerrail
      Contact( #AckRM10 )
   END_RUNG wire#w1
   RUNG wire#w2
      R_Coil( #Stop )
   END_RUNG
   RUNG wire#w2
      R_Coil( #Reset )
   END_RUNG
   RUNG wire#w2
      R_Coil( #StartConfirmationAck )
   END_RUNG
   RUNG wire#w2
      R_Coil( #EndConfirmationAck )
   END_RUNG
   RUNG wire#w2
      R_Coil( #AckRM1 )
   END_RUNG
   RUNG wire#w2
      R_Coil( #AckRM2 )
   END_RUNG
   RUNG wire#w2
      R_Coil( #AckRM3 )
   END_RUNG
   RUNG wire#w2
      R_Coil( #AckRM4 )
   END_RUNG
   RUNG wire#w2
      R_Coil( #AckRM5 )
   END_RUNG
   RUNG wire#w2
      R_Coil( #AckRM6 )
   END_RUNG
   RUNG wire#w2
      R_Coil( #AckRM7 )
   END_RUNG
   RUNG wire#w2
      R_Coil( #AckRM8 )
   END_RUNG
   RUNG wire#w2
      R_Coil( #AckRM9 )
   END_RUNG
   RUNG wire#w2
      R_Coil( #AckRM10 )
   END_RUNG
   // the same network as SCL:
   #BtnResetTimer(IN := #Start OR #Stop OR #Reset OR #StartConfirmationAck OR #EndConfirmationAck OR #AckRM1 OR #AckRM2 OR #AckRM3 OR #AckRM4 OR #AckRM5 OR #AckRM6 OR #AckRM7 OR #AckRM8 OR #AckRM9 OR #AckRM10,   // TON
                  PT := T#1s);
   IF #BtnResetTimer.Q THEN
       #Start := FALSE;
       #Stop := FALSE;
       #Reset := FALSE;
       #StartConfirmationAck := FALSE;
       #EndConfirmationAck := FALSE;
       #AckRM1 := FALSE;
       #AckRM2 := FALSE;
       #AckRM3 := FALSE;
       #AckRM4 := FALSE;
       #AckRM5 := FALSE;
       #AckRM6 := FALSE;
       #AckRM7 := FALSE;
       #AckRM8 := FALSE;
       #AckRM9 := FALSE;
       #AckRM10 := FALSE;
   END_IF;
END_REGION

REGION Network 11: Reset
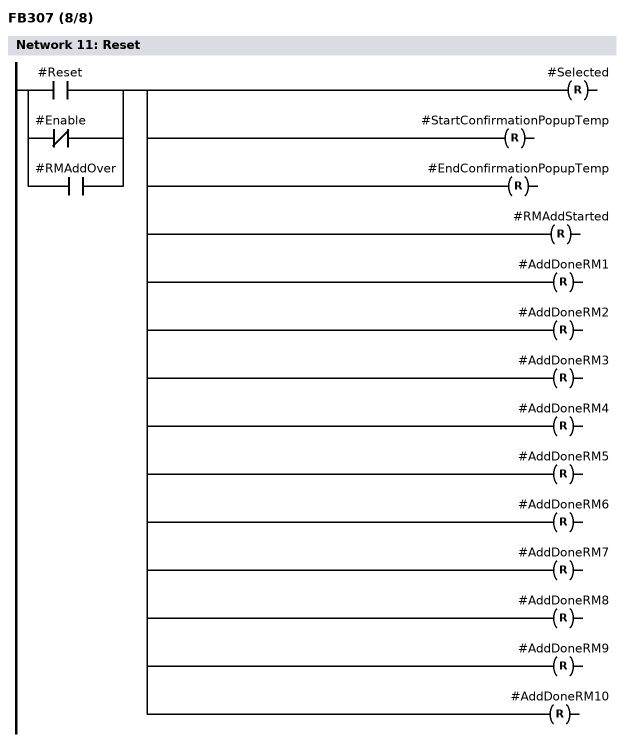
   RUNG wire#powerrail
      Contact( #Reset )
      wire#w1
      R_Coil( #Selected )
   END_RUNG
   RUNG wire#powerrail
      I_Contact( #Enable )
   END_RUNG wire#w1
   RUNG wire#powerrail
      Contact( #RMAddOver )
   END_RUNG wire#w1
   RUNG wire#w1
      R_Coil( #StartConfirmationPopupTemp )
   END_RUNG
   RUNG wire#w1
      R_Coil( #EndConfirmationPopupTemp )
   END_RUNG
   RUNG wire#w1
      R_Coil( #RMAddStarted )
   END_RUNG
   RUNG wire#w1
      R_Coil( #AddDoneRM1 )
   END_RUNG
   RUNG wire#w1
      R_Coil( #AddDoneRM2 )
   END_RUNG
   RUNG wire#w1
      R_Coil( #AddDoneRM3 )
   END_RUNG
   RUNG wire#w1
      R_Coil( #AddDoneRM4 )
   END_RUNG
   RUNG wire#w1
      R_Coil( #AddDoneRM5 )
   END_RUNG
   RUNG wire#w1
      R_Coil( #AddDoneRM6 )
   END_RUNG
   RUNG wire#w1
      R_Coil( #AddDoneRM7 )
   END_RUNG
   RUNG wire#w1
      R_Coil( #AddDoneRM8 )
   END_RUNG
   RUNG wire#w1
      R_Coil( #AddDoneRM9 )
   END_RUNG
   RUNG wire#w1
      R_Coil( #AddDoneRM10 )
   END_RUNG
   // the same network as SCL:
   IF #Reset OR NOT #Enable OR #RMAddOver THEN
       #Selected := FALSE;
       #StartConfirmationPopupTemp := FALSE;
       #EndConfirmationPopupTemp := FALSE;
       #RMAddStarted := FALSE;
       #AddDoneRM1 := FALSE;
       #AddDoneRM2 := FALSE;
       #AddDoneRM3 := FALSE;
       #AddDoneRM4 := FALSE;
       #AddDoneRM5 := FALSE;
       #AddDoneRM6 := FALSE;
       #AddDoneRM7 := FALSE;
       #AddDoneRM8 := FALSE;
       #AddDoneRM9 := FALSE;
       #AddDoneRM10 := FALSE;
   END_IF;
END_REGION
END_FUNCTION_BLOCK
